PROGRAM MAIN
VAR
	bStart			:BOOL;
	iStep			:INT;
	bCondition1 	:BOOL;
	bCondition2		:BOOL;
	bCondition3     :BOOL;
END_VAR

CASE iStep OF

	0: IF bStart THEN
		iStep:=10;
	   END_IF
	   
	10: IF bCondition1 THEN
		iStep:=0;
	    END_IF
END_CASE

END_PROGRAM

(* stored: Version 1.1.0.1, ProductVersion 3.1.4024.6
   POU MAIN: Id {7a32f106-3942-4996-95db-32d556c79356}, SpecialFunc None *)
